SUBAPPLICATION Uebung_009_AX (* Ticker *)
  (* Standard: 61499-2; Description: Copyright (c) 2023 Meisterschulen am Ostbahnhof This program and the accompanying materials are made available under the terms of the Eclipse Public License 2.0 which is available at https://www.eclipse.org/legal/epl-2.0/ SPDX-License-Identifier: EPL-2.0 *)
  (* Version 1.0, 2023-10-23, Franz Höpfinger, Meisterschulen am Ostbahnhof, initial API and implementation and/or initial documentation *)
  PACKAGE Uebungen;
  IMPORT Uebungen::const::UT::DefaultPool::OutputNumber_N1;
  IMPORT logiBUS::io::DQ::logiBUS_DO::Output_Q1;
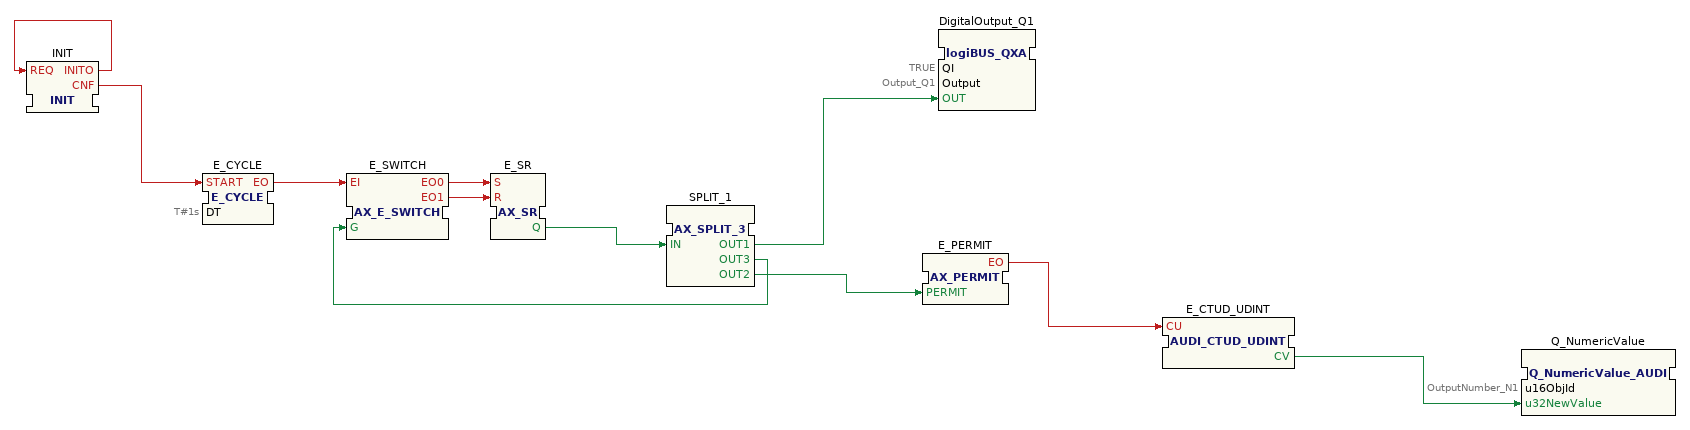
  FBS
    DigitalOutput_Q1 : logiBUS::io::DQ::logiBUS_QXA(QI := TRUE, Output := Output_Q1);
    E_CYCLE : iec61499::events::E_CYCLE(DT := T#1s);
    E_SWITCH : adapter::events::unidirectional::AX_E_SWITCH;
    E_SR : adapter::events::unidirectional::AX_SR;
    E_PERMIT : adapter::events::unidirectional::AX_PERMIT;
    E_CTUD_UDINT : adapter::events::unidirectional::AUDI_CTUD_UDINT;
    Q_NumericValue : isobus::UT::Q::Q_NumericValue_AUDI(u16ObjId := OutputNumber_N1);
    INIT : iec61131::booleanOperators::INIT;
    SPLIT_1 : adapter::events::unidirectional::AX_SPLIT_3;
  END_FBS
  EVENT_CONNECTIONS
    E_CYCLE.EO TO E_SWITCH.EI;
    E_SWITCH.EO0 TO E_SR.S;
    E_SWITCH.EO1 TO E_SR.R;
    E_PERMIT.EO TO E_CTUD_UDINT.CU;
    INIT.INITO TO INIT.REQ;
    INIT.CNF TO E_CYCLE.START;
  END_CONNECTIONS
  ADAPTER_CONNECTIONS
    SPLIT_1.OUT1 TO DigitalOutput_Q1.OUT;
    E_SR.Q TO SPLIT_1.IN;
    SPLIT_1.OUT3 TO E_SWITCH.G;
    SPLIT_1.OUT2 TO E_PERMIT.PERMIT;
    E_CTUD_UDINT.CV TO Q_NumericValue.u32NewValue;
  END_CONNECTIONS
END_SUBAPPLICATION
